Staubli VAL3: countItem.dtx

public bool bActive
public string sID
public string sName
public num nCount
public bool bEnable
